ABB RAPID module: Module1.mod

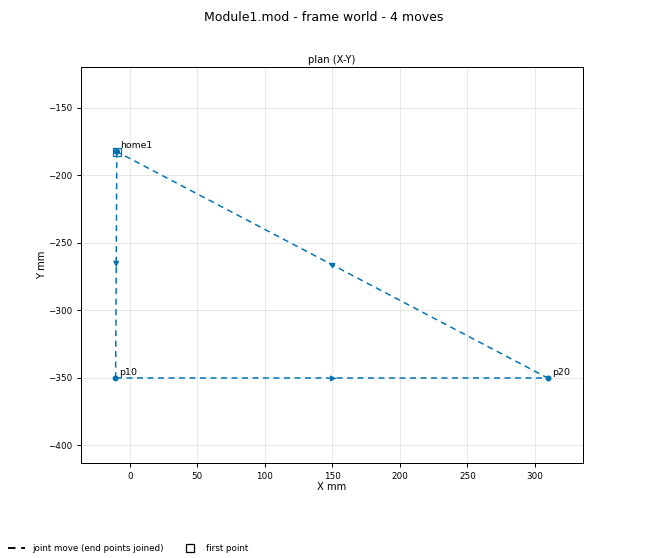
[picture p0: tool path of Module1.mod in frame world, 4 of 4 moves have a stored position in this frame; points joined in program order, loops and branches not executed]
MODULE Module1
	CONST robtarget p10:=[[-10.44,-350.54,199.40],[0.0629343,-0.843397,-0.111239,-0.521869],[0,0,0,4],[-101.614,9E+9,9E+9,9E+9,9E+9,9E+9]];
	CONST robtarget p20:=[[310.13,-350.54,199.40],[0.0629343,-0.843397,-0.111239,-0.521869],[1,-1,1,4],[-101.614,9E+9,9E+9,9E+9,9E+9,9E+9]];
	CONST robtarget home:=[[-9.58,-182.61,198.63],[0.0660107,-0.842421,-0.111215,-0.523069],[0,0,0,4],[-101.964,9E+9,9E+9,9E+9,9E+9,9E+9]];
	CONST robtarget home1:=[[-9.58,-182.61,198.63],[0.0660107,-0.842421,-0.111215,-0.523069],[0,0,0,4],[-101.964,9E+9,9E+9,9E+9,9E+9,9E+9]];
	CONST robtarget home11:=[[-9.58,-182.61,198.63],[0.0660107,-0.842421,-0.111215,-0.523069],[0,0,0,4],[-101.964,9E+9,9E+9,9E+9,9E+9,9E+9]];
	CONST robtarget p30:=[[310.13,-350.54,199.40],[0.0629343,-0.843397,-0.111239,-0.521869],[1,-1,1,4],[-101.614,9E+9,9E+9,9E+9,9E+9,9E+9]];
    !***********************************************************
    !
    ! Module:  Module1
    !
    ! Description:
    !   <Insert description here>
    !
    ! Author: anasm
    !
    ! Version: 1.0
    !
    !***********************************************************


    !***********************************************************
    !
    ! Procedure main
    !
    !   This is the entry point of your program
    !
    !***********************************************************
    PROC main()
        !Add your code here
        MoveJ home1, v1000, z50, tool0;
        MoveJ p10, v1000, z50, tool0;
        WaitTime 1;
        MoveJ p20, v1000, z50, tool0;
        WaitTime 1;
        MoveJ home1, v1000, z50, tool0;
    ENDPROC
ENDMODULE
